(* Logix 5000 project; controller cal1632 1756-L62 rev 16.20; software revision 16.05; part 43 of 57 *)
(* tags used below, declared in another part *)
   FAULT : BOOL;
   HMI : BOOL;
   p01_recipe_active : recipe;
   p01r02_plc_scan_time_in_sec : REAL;
   p01r09_pb_global_reset : BOOL;
   p01r09_request_line_jog : BOOL;
   p01r09_stretch_mode : BOOL;
   p01r12_master_ramped_speed : REAL;
   p01r13_line_running : BOOL;
   p01r13_line_slow_ramp : BOOL;
   p01r13_permissive_drives : BOOL;
   p01r13_state : DINT;
   p02_real_from_hmi : hmi_real;
   p20r15_loa_on : BOOL;
   p20r16_lob_on : BOOL;
   p22r09_mode_thread : BOOL;
   p22r10_pid_psn : PID;
   p25_ai_speed : REAL;
   p25_ai_torque : REAL;
   p25_ai_ts2_lc : REAL;
   p25_ao_selected_speed : REAL;
   p25_ao_torque : REAL;
   p25_control_word : INT;
   p25_di_brake : BOOL;
   p25_di_jog : BOOL;
   p25_di_jog_fwd : BOOL;
   p25_di_jog_rev : BOOL;
   p25_di_run : BOOL;
   p25_di_therm : BOOL;
   p25_dint_to_hmi : DINT[16];
   p25_param_ts2_jog_speed : REAL;
   p25_status_word : INT;
   p25_ts2_acc_rate : REAL;
   p25_ts2_decel_rate : REAL;
   p25_ts2_vfd : ABB_PROTOCOL_VFD;
   p25r02_tension_dev_max : REAL;
   p25r02_tension_dev_min : REAL;
   p25r08 : routine;
   p25r08_timer_fault : TIMER[4];
   p25r08_timer_warning : TIMER[4];
   p25r09 : routine;
   p25r09_mode_jog : BOOL;
   p25r09_mode_run : BOOL;
   p25r09_mode_thread : BOOL;
   p25r09_pb_jog_fwd : BOOL;
   p25r09_pb_jog_rev : BOOL;
   p25r09_timer_fault : TIMER[4];
   p25r09_timer_warning : TIMER[4];
   p25r10 : routine;
   p25r10_calc_speed_offset : REAL;
   p25r10_param_psn_gain : REAL;
   p25r10_pid_manual_request : BOOL;
   p25r10_pid_out : REAL;
   p25r10_pid_psn : PID;
   p25r10_pid_psn_cv : REAL;
   p25r10_pid_psn_pv : REAL;
   p25r10_speed_offset : REAL;
   p25r10_tension_request : BOOL;
   p25r10_timer_fault : TIMER[4];
   p25r10_timer_warning : TIMER[4];
   p25r11 : routine;
   p25r11_acc_decel_ramp : SYS_ACC_DEC_RAMP;
   p25r11_at_zero : BOOL;
   p25r11_permissive_jog_thread : BOOL;
   p25r11_request_jog_fwd : BOOL;
   p25r11_request_jog_rev : BOOL;
   p25r11_request_line_jog : BOOL;
   p25r11_request_line_run : BOOL;
   p25r11_request_thread_fwd : BOOL;
   p25r11_request_thread_rev : BOOL;
   p25r11_selected_speed : REAL;
   p25r11_timer_fault : TIMER[10];
   p25r11_timer_warning : TIMER[4];
   p25r11_vfd_start_request : BOOL;
(* P25_Tension_Stand_2, continued *)

ROUTINE R08_Warnings   (* ladder *)
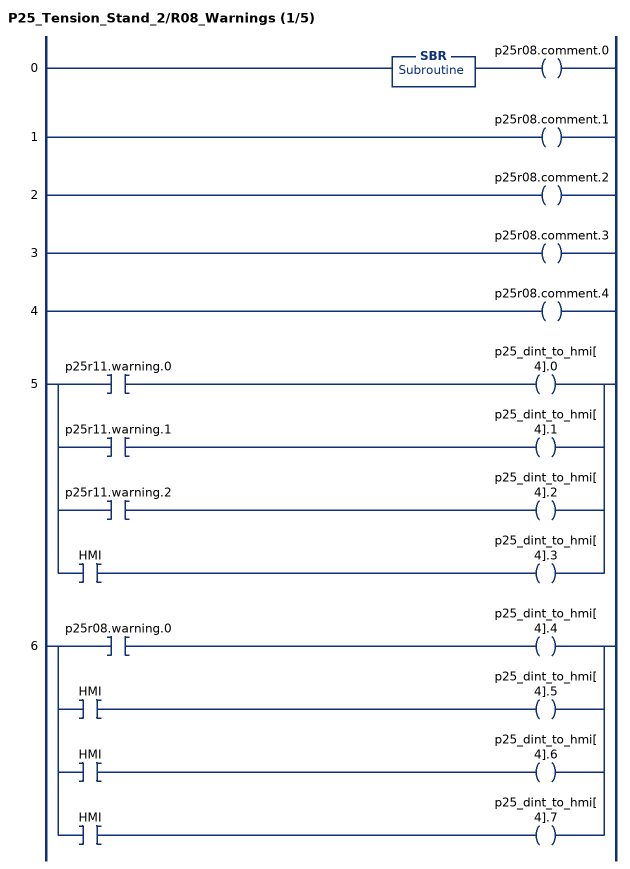
   0: SBR()OTE(p25r08.comment.0);
   1: OTE(p25r08.comment.1);
   2: OTE(p25r08.comment.2);
   3: OTE(p25r08.comment.3);
   4: OTE(p25r08.comment.4);
   5: [XIC(p25r11.warning.0) OTE(p25_dint_to_hmi[4].0) ,XIC(p25r11.warning.1) OTE(p25_dint_to_hmi[4].1) ,XIC(p25r11.warning.2) OTE(p25_dint_to_hmi[4].2) ,XIC(HMI) OTE(p25_dint_to_hmi[4].3) ];
   6: [XIC(p25r08.warning.0) OTE(p25_dint_to_hmi[4].4) ,XIC(HMI) OTE(p25_dint_to_hmi[4].5) ,XIC(HMI) OTE(p25_dint_to_hmi[4].6) ,XIC(HMI) OTE(p25_dint_to_hmi[4].7) ];
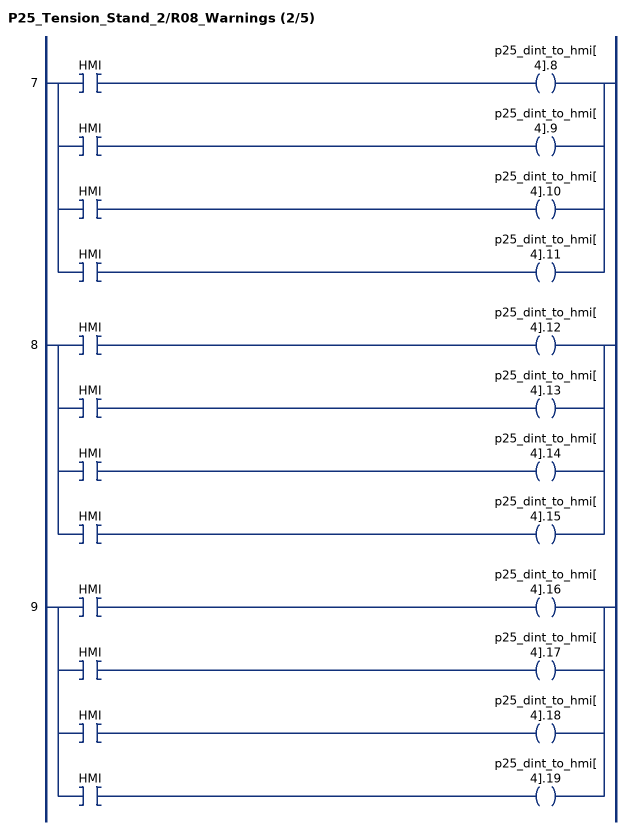
   7: [XIC(HMI) OTE(p25_dint_to_hmi[4].8) ,XIC(HMI) OTE(p25_dint_to_hmi[4].9) ,XIC(HMI) OTE(p25_dint_to_hmi[4].10) ,XIC(HMI) OTE(p25_dint_to_hmi[4].11) ];
   8: [XIC(HMI) OTE(p25_dint_to_hmi[4].12) ,XIC(HMI) OTE(p25_dint_to_hmi[4].13) ,XIC(HMI) OTE(p25_dint_to_hmi[4].14) ,XIC(HMI) OTE(p25_dint_to_hmi[4].15) ];
   9: [XIC(HMI) OTE(p25_dint_to_hmi[4].16) ,XIC(HMI) OTE(p25_dint_to_hmi[4].17) ,XIC(HMI) OTE(p25_dint_to_hmi[4].18) ,XIC(HMI) OTE(p25_dint_to_hmi[4].19) ];
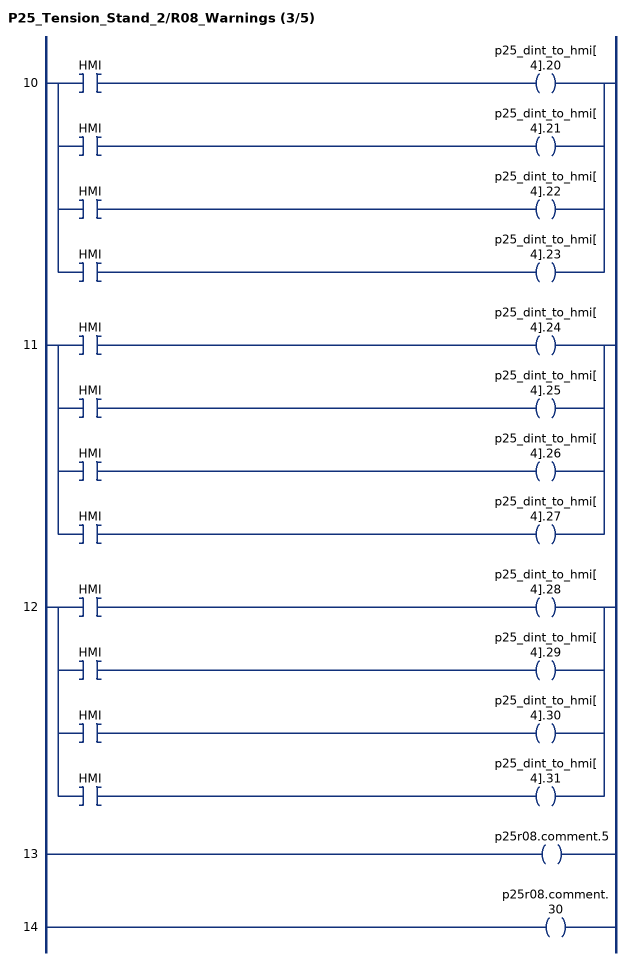
   10: [XIC(HMI) OTE(p25_dint_to_hmi[4].20) ,XIC(HMI) OTE(p25_dint_to_hmi[4].21) ,XIC(HMI) OTE(p25_dint_to_hmi[4].22) ,XIC(HMI) OTE(p25_dint_to_hmi[4].23) ];
   11: [XIC(HMI) OTE(p25_dint_to_hmi[4].24) ,XIC(HMI) OTE(p25_dint_to_hmi[4].25) ,XIC(HMI) OTE(p25_dint_to_hmi[4].26) ,XIC(HMI) OTE(p25_dint_to_hmi[4].27) ];
   12: [XIC(HMI) OTE(p25_dint_to_hmi[4].28) ,XIC(HMI) OTE(p25_dint_to_hmi[4].29) ,XIC(HMI) OTE(p25_dint_to_hmi[4].30) ,XIC(HMI) OTE(p25_dint_to_hmi[4].31) ];
   13: OTE(p25r08.comment.5);
   14: OTE(p25r08.comment.30);
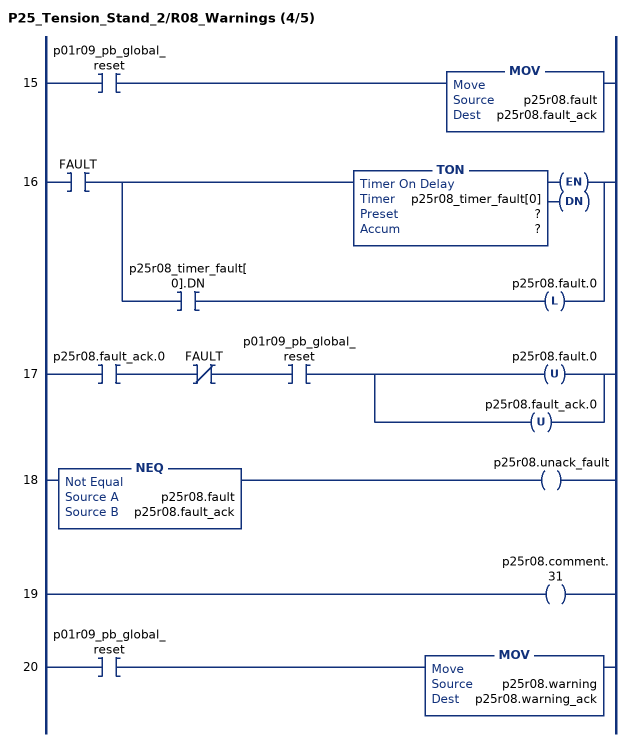
   15: XIC(p01r09_pb_global_reset)MOV(p25r08.fault,p25r08.fault_ack);
   16: XIC(FAULT)[TON(p25r08_timer_fault[0],?,?) ,XIC(p25r08_timer_fault[0].DN) OTL(p25r08.fault.0) ];
   17: XIC(p25r08.fault_ack.0)XIO(FAULT)XIC(p01r09_pb_global_reset)[OTU(p25r08.fault.0) ,OTU(p25r08.fault_ack.0) ];
   18: NEQ(p25r08.fault,p25r08.fault_ack)OTE(p25r08.unack_fault);
   19: OTE(p25r08.comment.31);
   20: XIC(p01r09_pb_global_reset)MOV(p25r08.warning,p25r08.warning_ack);
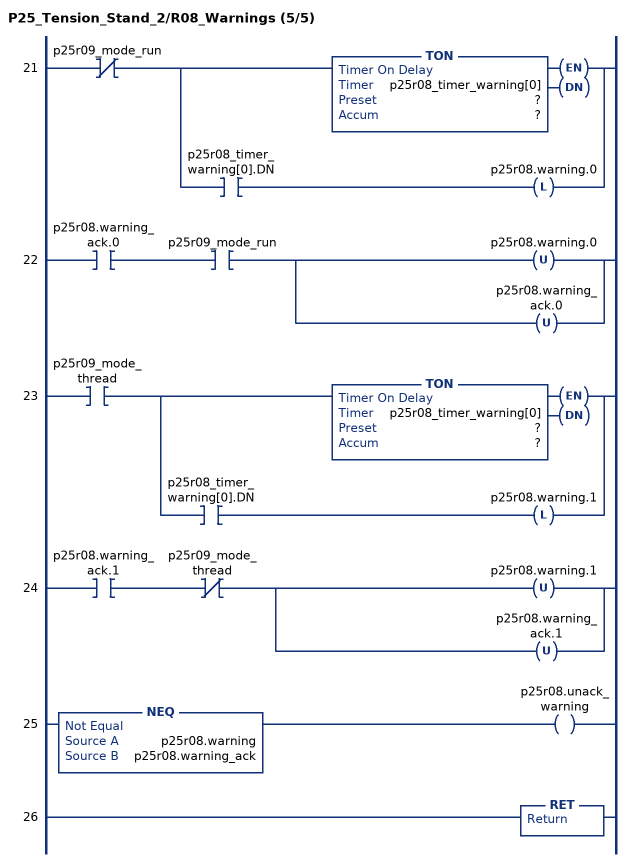
   21: XIO(p25r09_mode_run)[TON(p25r08_timer_warning[0],?,?) ,XIC(p25r08_timer_warning[0].DN) OTL(p25r08.warning.0) ];
   22: XIC(p25r08.warning_ack.0)XIC(p25r09_mode_run)[OTU(p25r08.warning.0) ,OTU(p25r08.warning_ack.0) ];
   23: XIC(p25r09_mode_thread)[TON(p25r08_timer_warning[0],?,?) ,XIC(p25r08_timer_warning[0].DN) OTL(p25r08.warning.1) ];
   24: XIC(p25r08.warning_ack.1)XIO(p25r09_mode_thread)[OTU(p25r08.warning.1) ,OTU(p25r08.warning_ack.1) ];
   25: NEQ(p25r08.warning,p25r08.warning_ack)OTE(p25r08.unack_warning);
   26: RET();
END_ROUTINE

ROUTINE R09_Modes   (* ladder *)
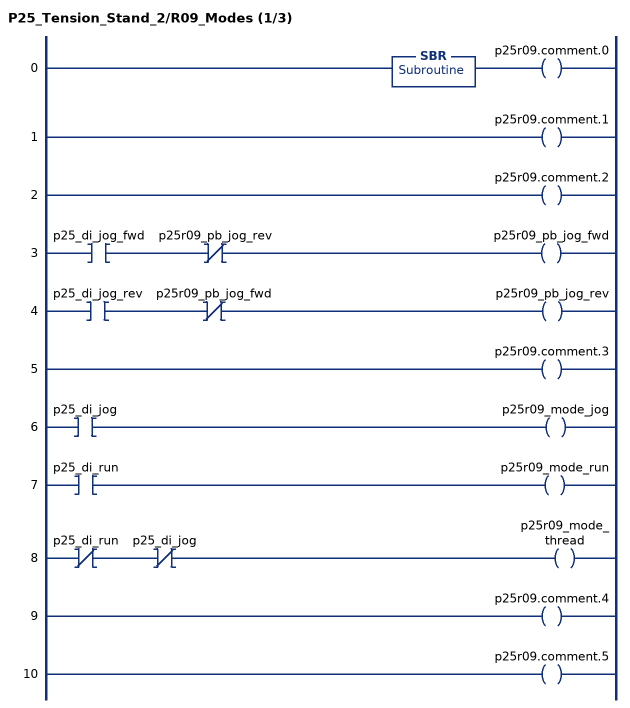
   0: SBR()OTE(p25r09.comment.0);
   1: OTE(p25r09.comment.1);
   2: OTE(p25r09.comment.2);
   3: XIC(p25_di_jog_fwd)XIO(p25r09_pb_jog_rev)OTE(p25r09_pb_jog_fwd);
   4: XIC(p25_di_jog_rev)XIO(p25r09_pb_jog_fwd)OTE(p25r09_pb_jog_rev);
   5: OTE(p25r09.comment.3);
   6: XIC(p25_di_jog)OTE(p25r09_mode_jog);
   7: XIC(p25_di_run)OTE(p25r09_mode_run);
   8: XIO(p25_di_run)XIO(p25_di_jog)OTE(p25r09_mode_thread);
   9: OTE(p25r09.comment.4);
   10: OTE(p25r09.comment.5);
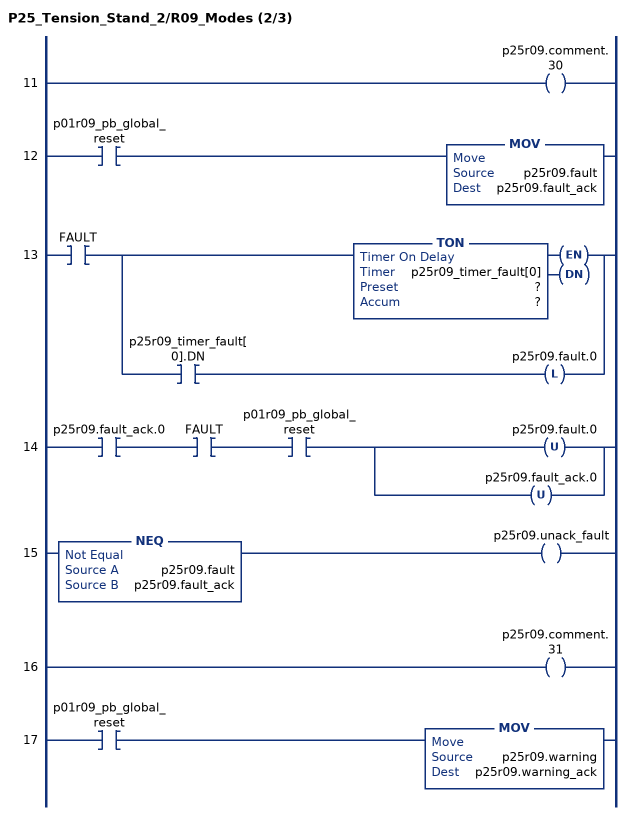
   11: OTE(p25r09.comment.30);
   12: XIC(p01r09_pb_global_reset)MOV(p25r09.fault,p25r09.fault_ack);
   13: XIC(FAULT)[TON(p25r09_timer_fault[0],?,?) ,XIC(p25r09_timer_fault[0].DN) OTL(p25r09.fault.0) ];
   14: XIC(p25r09.fault_ack.0)XIC(FAULT)XIC(p01r09_pb_global_reset)[OTU(p25r09.fault.0) ,OTU(p25r09.fault_ack.0) ];
   15: NEQ(p25r09.fault,p25r09.fault_ack)OTE(p25r09.unack_fault);
   16: OTE(p25r09.comment.31);
   17: XIC(p01r09_pb_global_reset)MOV(p25r09.warning,p25r09.warning_ack);
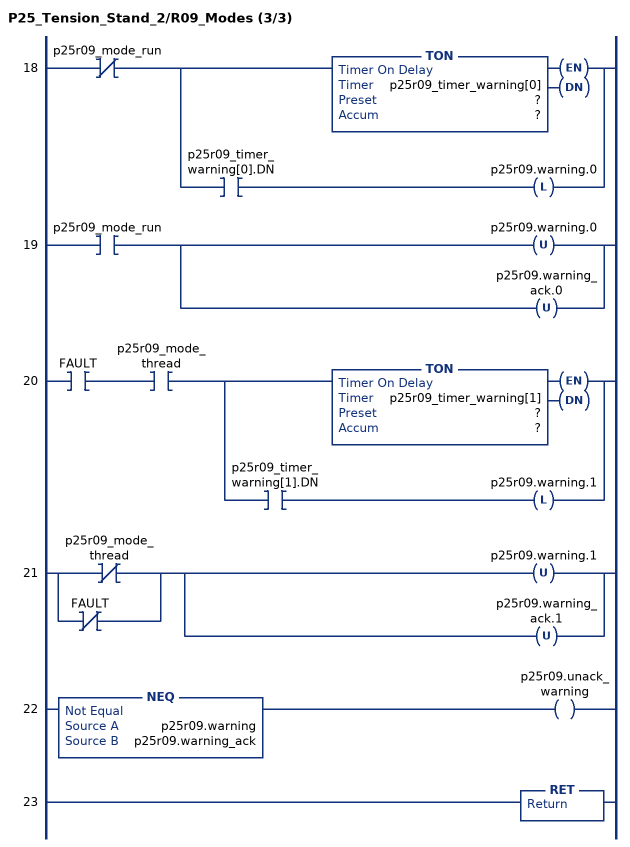
   18: XIO(p25r09_mode_run)[TON(p25r09_timer_warning[0],?,?) ,XIC(p25r09_timer_warning[0].DN) OTL(p25r09.warning.0) ];
   19: XIC(p25r09_mode_run)[OTU(p25r09.warning.0) ,OTU(p25r09.warning_ack.0) ];
   20: XIC(FAULT)XIC(p25r09_mode_thread)[TON(p25r09_timer_warning[1],?,?) ,XIC(p25r09_timer_warning[1].DN) OTL(p25r09.warning.1) ];
   21: [XIO(p25r09_mode_thread) ,XIO(FAULT) ][OTU(p25r09.warning.1) ,OTU(p25r09.warning_ack.1) ];
   22: NEQ(p25r09.warning,p25r09.warning_ack)OTE(p25r09.unack_warning);
   23: RET();
END_ROUTINE

ROUTINE R10_Speed_Control   (* ladder *)
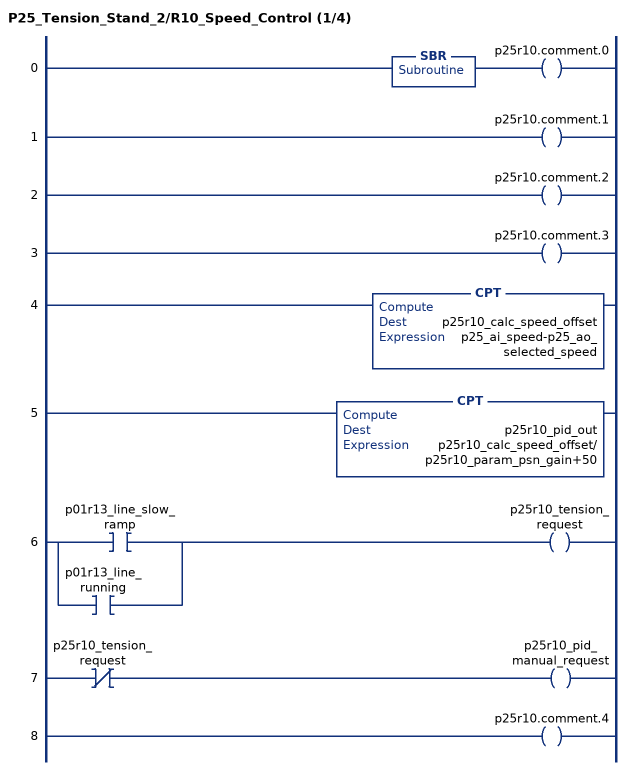
   0: SBR()OTE(p25r10.comment.0);
   1: OTE(p25r10.comment.1);
   2: OTE(p25r10.comment.2);
   3: OTE(p25r10.comment.3);
   4: CPT(p25r10_calc_speed_offset,p25_ai_speed-p25_ao_selected_speed);
   5: CPT(p25r10_pid_out,p25r10_calc_speed_offset/p25r10_param_psn_gain+50);
   6: [XIC(p01r13_line_slow_ramp) ,XIC(p01r13_line_running) ]OTE(p25r10_tension_request);
   7: XIO(p25r10_tension_request)OTE(p25r10_pid_manual_request);
   8: OTE(p25r10.comment.4);
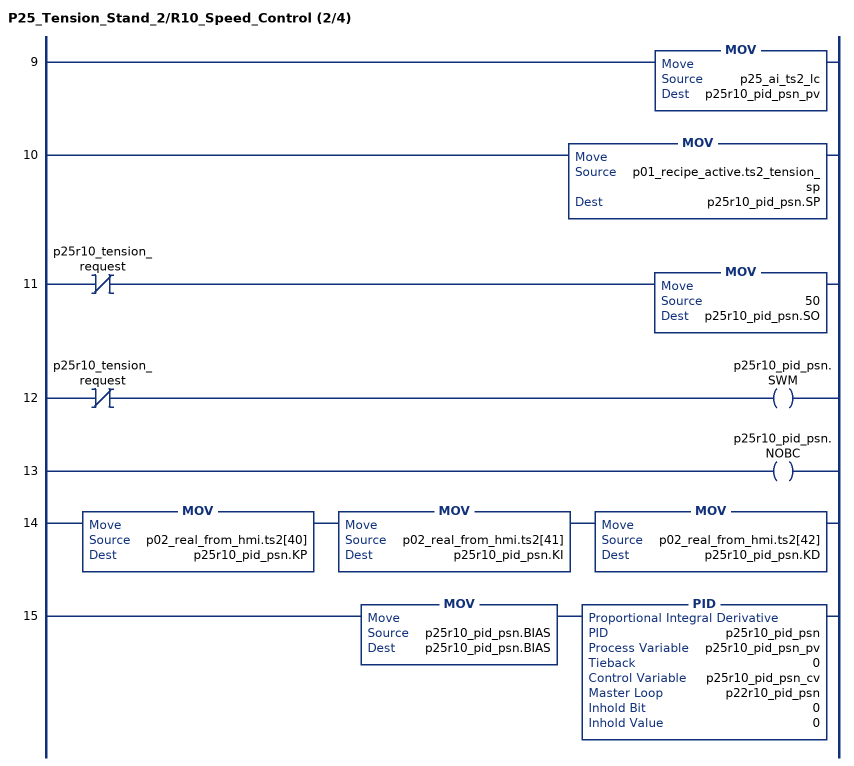
   9: MOV(p25_ai_ts2_lc,p25r10_pid_psn_pv);
   10: MOV(p01_recipe_active.ts2_tension_sp,p25r10_pid_psn.SP);
   11: XIO(p25r10_tension_request)MOV(50,p25r10_pid_psn.SO);
   12: XIO(p25r10_tension_request)OTE(p25r10_pid_psn.SWM);
   13: OTE(p25r10_pid_psn.NOBC);
   14: MOV(p02_real_from_hmi.ts2[40],p25r10_pid_psn.KP)MOV(p02_real_from_hmi.ts2[41],p25r10_pid_psn.KI)MOV(p02_real_from_hmi.ts2[42],p25r10_pid_psn.KD);
   15: MOV(p25r10_pid_psn.BIAS,p25r10_pid_psn.BIAS)PID(p25r10_pid_psn,p25r10_pid_psn_pv,0,p25r10_pid_psn_cv,p22r10_pid_psn,0,0);
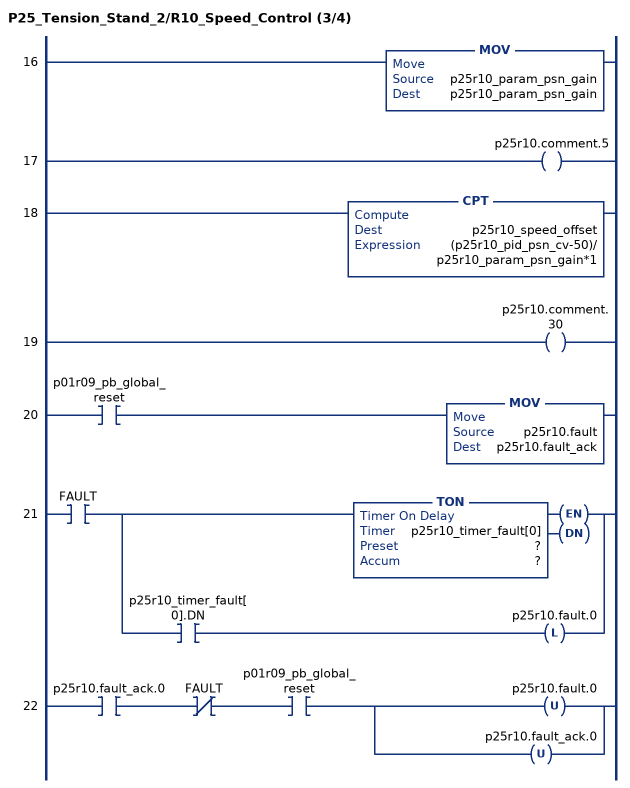
   16: MOV(p25r10_param_psn_gain,p25r10_param_psn_gain);
   17: OTE(p25r10.comment.5);
   18: CPT(p25r10_speed_offset,(p25r10_pid_psn_cv-50)/p25r10_param_psn_gain*1);
   19: OTE(p25r10.comment.30);
   20: XIC(p01r09_pb_global_reset)MOV(p25r10.fault,p25r10.fault_ack);
   21: XIC(FAULT)[TON(p25r10_timer_fault[0],?,?) ,XIC(p25r10_timer_fault[0].DN) OTL(p25r10.fault.0) ];
   22: XIC(p25r10.fault_ack.0)XIO(FAULT)XIC(p01r09_pb_global_reset)[OTU(p25r10.fault.0) ,OTU(p25r10.fault_ack.0) ];
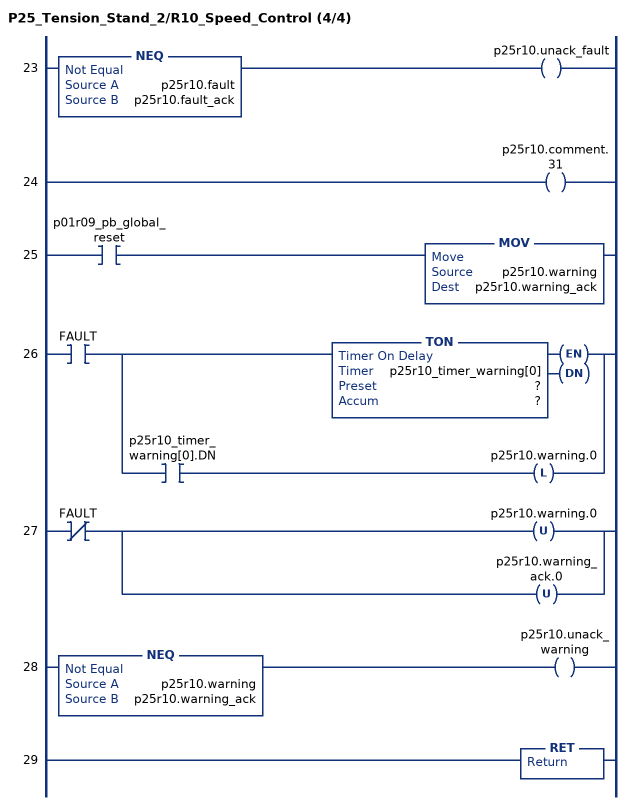
   23: NEQ(p25r10.fault,p25r10.fault_ack)OTE(p25r10.unack_fault);
   24: OTE(p25r10.comment.31);
   25: XIC(p01r09_pb_global_reset)MOV(p25r10.warning,p25r10.warning_ack);
   26: XIC(FAULT)[TON(p25r10_timer_warning[0],?,?) ,XIC(p25r10_timer_warning[0].DN) OTL(p25r10.warning.0) ];
   27: XIO(FAULT)[OTU(p25r10.warning.0) ,OTU(p25r10.warning_ack.0) ];
   28: NEQ(p25r10.warning,p25r10.warning_ack)OTE(p25r10.unack_warning);
   29: RET();
END_ROUTINE

ROUTINE R11_VFD   (* ladder *)
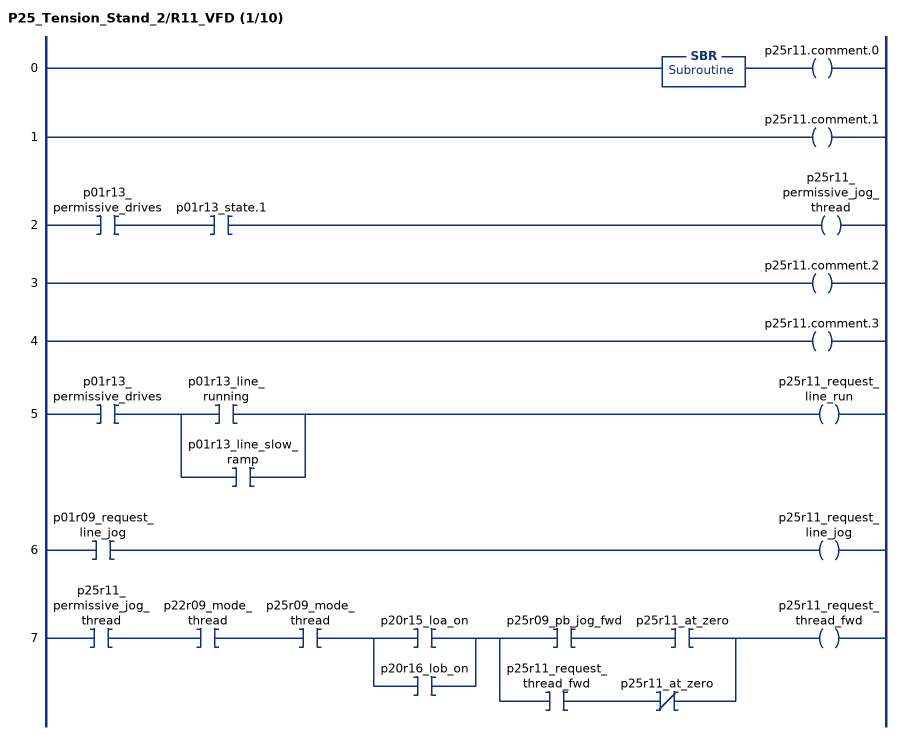
   0: SBR()OTE(p25r11.comment.0);
   1: OTE(p25r11.comment.1);
   2: XIC(p01r13_permissive_drives)XIC(p01r13_state.1)OTE(p25r11_permissive_jog_thread);
   3: OTE(p25r11.comment.2);
   4: OTE(p25r11.comment.3);
   5: XIC(p01r13_permissive_drives)[XIC(p01r13_line_running) ,XIC(p01r13_line_slow_ramp) ]OTE(p25r11_request_line_run);
   6: XIC(p01r09_request_line_jog)OTE(p25r11_request_line_jog);
   7: XIC(p25r11_permissive_jog_thread)XIC(p22r09_mode_thread)XIC(p25r09_mode_thread)[XIC(p20r15_loa_on) ,XIC(p20r16_lob_on) ][XIC(p25r09_pb_jog_fwd) XIC(p25r11_at_zero) ,XIC(p25r11_request_thread_fwd) XIO(p25r11_at_zero) ]OTE(p25r11_request_thread_fwd);
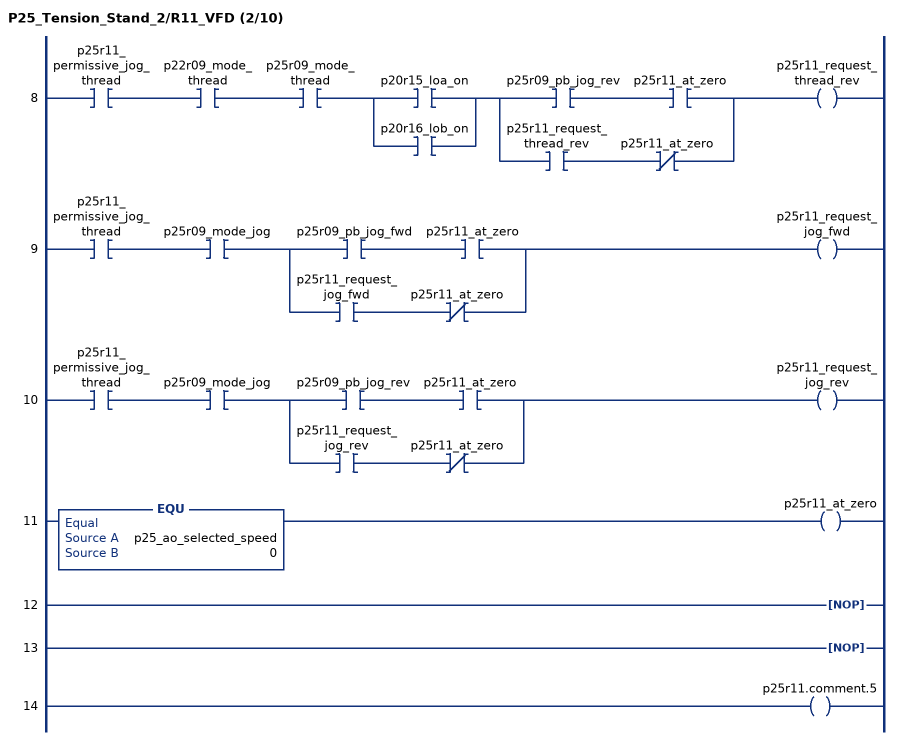
   8: XIC(p25r11_permissive_jog_thread)XIC(p22r09_mode_thread)XIC(p25r09_mode_thread)[XIC(p20r15_loa_on) ,XIC(p20r16_lob_on) ][XIC(p25r09_pb_jog_rev) XIC(p25r11_at_zero) ,XIC(p25r11_request_thread_rev) XIO(p25r11_at_zero) ]OTE(p25r11_request_thread_rev);
   9: XIC(p25r11_permissive_jog_thread)XIC(p25r09_mode_jog)[XIC(p25r09_pb_jog_fwd) XIC(p25r11_at_zero) ,XIC(p25r11_request_jog_fwd) XIO(p25r11_at_zero) ]OTE(p25r11_request_jog_fwd);
   10: XIC(p25r11_permissive_jog_thread)XIC(p25r09_mode_jog)[XIC(p25r09_pb_jog_rev) XIC(p25r11_at_zero) ,XIC(p25r11_request_jog_rev) XIO(p25r11_at_zero) ]OTE(p25r11_request_jog_rev);
   11: EQU(p25_ao_selected_speed,0)OTE(p25r11_at_zero);
   12: NOP();
   13: NOP();
   14: OTE(p25r11.comment.5);
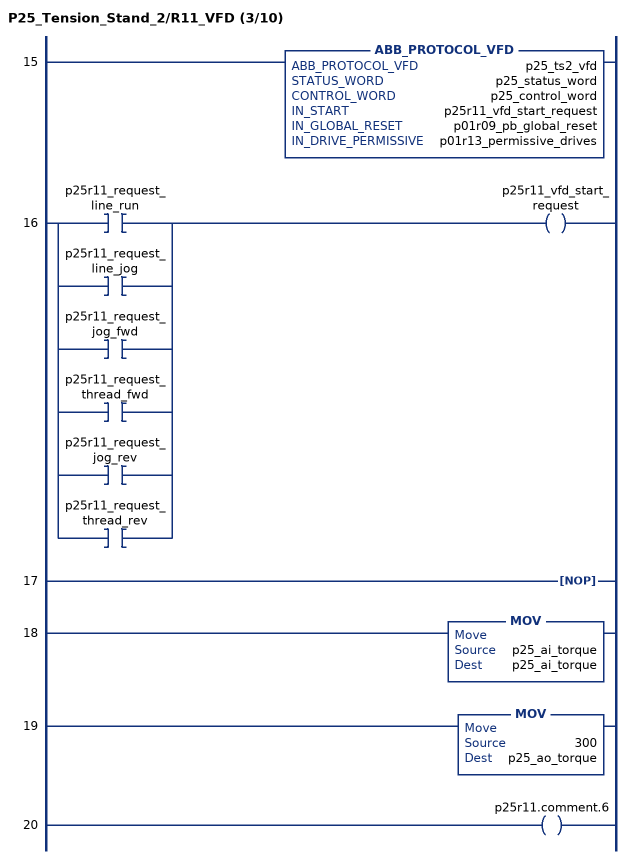
   15: ABB_PROTOCOL_VFD(p25_ts2_vfd,p25_status_word,p25_control_word,p25r11_vfd_start_request,p01r09_pb_global_reset,p01r13_permissive_drives);
   16: [XIC(p25r11_request_line_run) ,XIC(p25r11_request_line_jog) ,XIC(p25r11_request_jog_fwd) ,XIC(p25r11_request_thread_fwd) ,XIC(p25r11_request_jog_rev) ,XIC(p25r11_request_thread_rev) ]OTE(p25r11_vfd_start_request);
   17: NOP();
   18: MOV(p25_ai_torque,p25_ai_torque);
   19: MOV(300,p25_ao_torque);
   20: OTE(p25r11.comment.6);
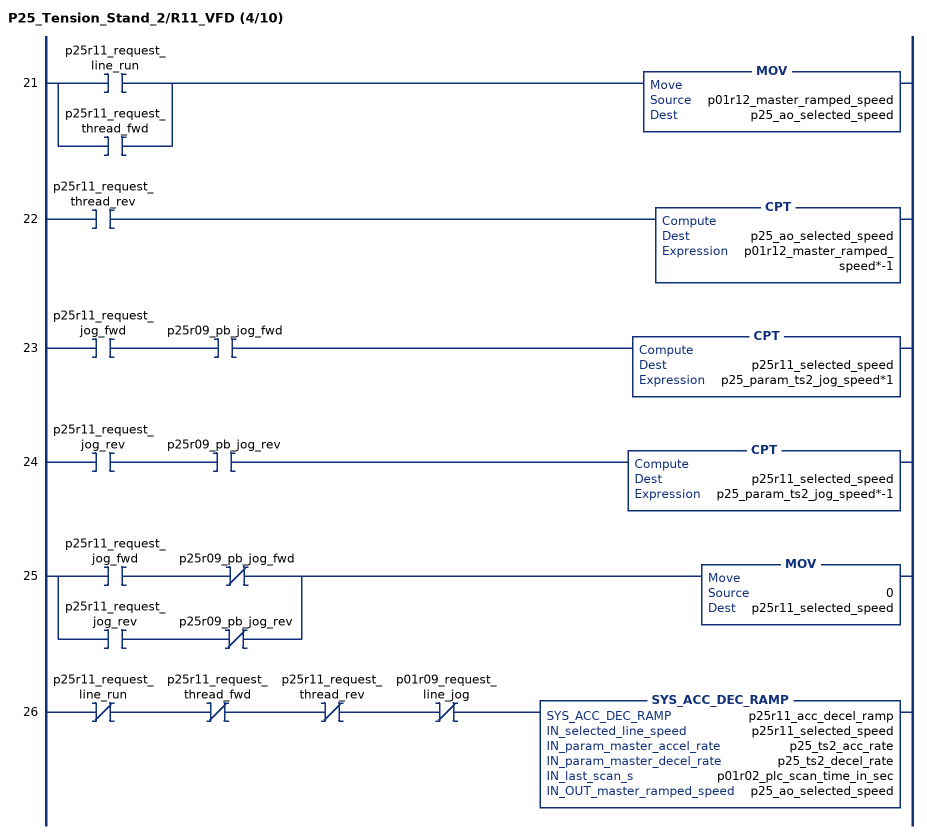
   21: [XIC(p25r11_request_line_run) ,XIC(p25r11_request_thread_fwd) ]MOV(p01r12_master_ramped_speed,p25_ao_selected_speed);
   22: XIC(p25r11_request_thread_rev)CPT(p25_ao_selected_speed,p01r12_master_ramped_speed*-1);
   23: XIC(p25r11_request_jog_fwd)XIC(p25r09_pb_jog_fwd)CPT(p25r11_selected_speed,p25_param_ts2_jog_speed*1);
   24: XIC(p25r11_request_jog_rev)XIC(p25r09_pb_jog_rev)CPT(p25r11_selected_speed,p25_param_ts2_jog_speed*-1);
   25: [XIC(p25r11_request_jog_fwd) XIO(p25r09_pb_jog_fwd) ,XIC(p25r11_request_jog_rev) XIO(p25r09_pb_jog_rev) ]MOV(0,p25r11_selected_speed);
   26: XIO(p25r11_request_line_run)XIO(p25r11_request_thread_fwd)XIO(p25r11_request_thread_rev)XIO(p01r09_request_line_jog)SYS_ACC_DEC_RAMP(p25r11_acc_decel_ramp,p25r11_selected_speed,p25_ts2_acc_rate,p25_ts2_decel_rate,p01r02_plc_scan_time_in_sec,p25_ao_selected_speed);
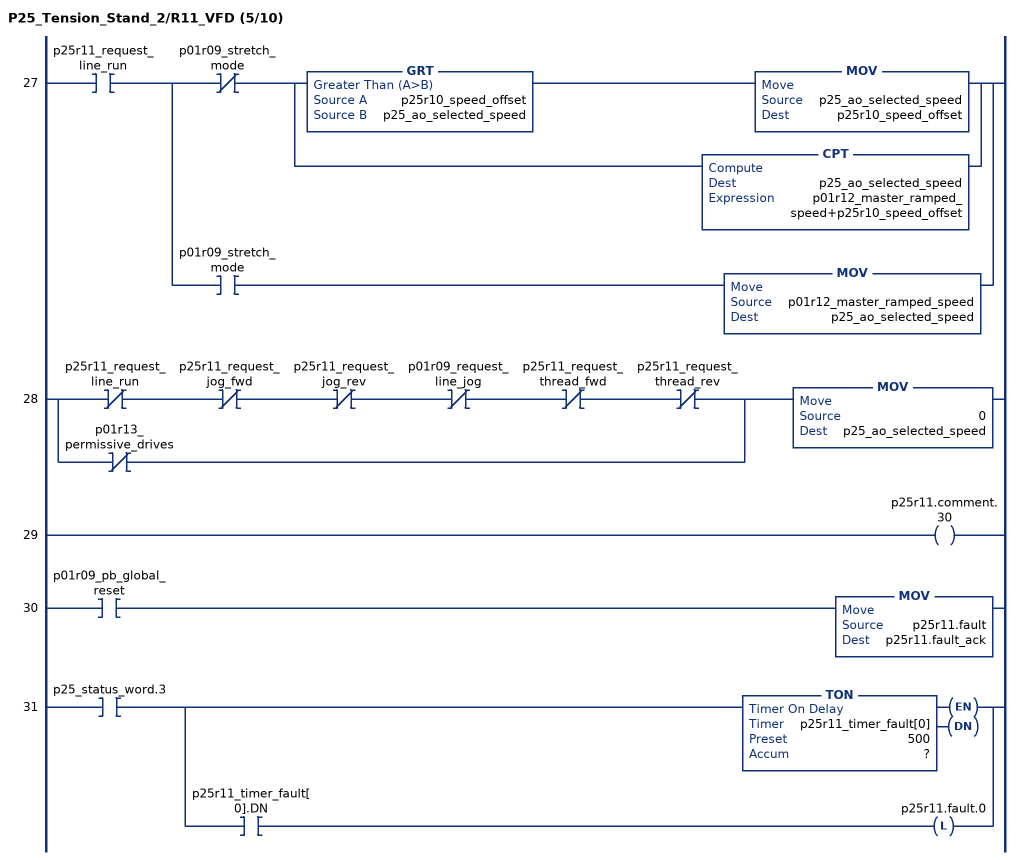
   27: XIC(p25r11_request_line_run)[XIO(p01r09_stretch_mode) [GRT(p25r10_speed_offset,p25_ao_selected_speed) MOV(p25_ao_selected_speed,p25r10_speed_offset) ,CPT(p25_ao_selected_speed,p01r12_master_ramped_speed+p25r10_speed_offset) ] ,XIC(p01r09_stretch_mode) MOV(p01r12_master_ramped_speed,p25_ao_selected_speed) ];
   28: [XIO(p25r11_request_line_run) XIO(p25r11_request_jog_fwd) XIO(p25r11_request_jog_rev) XIO(p01r09_request_line_jog) XIO(p25r11_request_thread_fwd) XIO(p25r11_request_thread_rev) ,XIO(p01r13_permissive_drives) ]MOV(0,p25_ao_selected_speed);
   29: OTE(p25r11.comment.30);
   30: XIC(p01r09_pb_global_reset)MOV(p25r11.fault,p25r11.fault_ack);
   31: XIC(p25_status_word.3)[TON(p25r11_timer_fault[0],?,?) ,XIC(p25r11_timer_fault[0].DN) OTL(p25r11.fault.0) ];
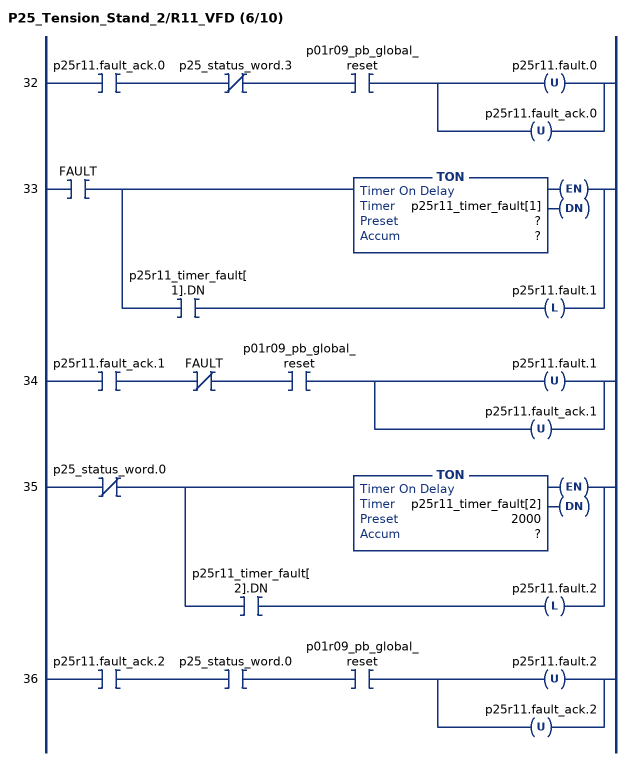
   32: XIC(p25r11.fault_ack.0)XIO(p25_status_word.3)XIC(p01r09_pb_global_reset)[OTU(p25r11.fault.0) ,OTU(p25r11.fault_ack.0) ];
   33: XIC(FAULT)[TON(p25r11_timer_fault[1],?,?) ,XIC(p25r11_timer_fault[1].DN) OTL(p25r11.fault.1) ];
   34: XIC(p25r11.fault_ack.1)XIO(FAULT)XIC(p01r09_pb_global_reset)[OTU(p25r11.fault.1) ,OTU(p25r11.fault_ack.1) ];
   35: XIO(p25_status_word.0)[TON(p25r11_timer_fault[2],?,?) ,XIC(p25r11_timer_fault[2].DN) OTL(p25r11.fault.2) ];
   36: XIC(p25r11.fault_ack.2)XIC(p25_status_word.0)XIC(p01r09_pb_global_reset)[OTU(p25r11.fault.2) ,OTU(p25r11.fault_ack.2) ];
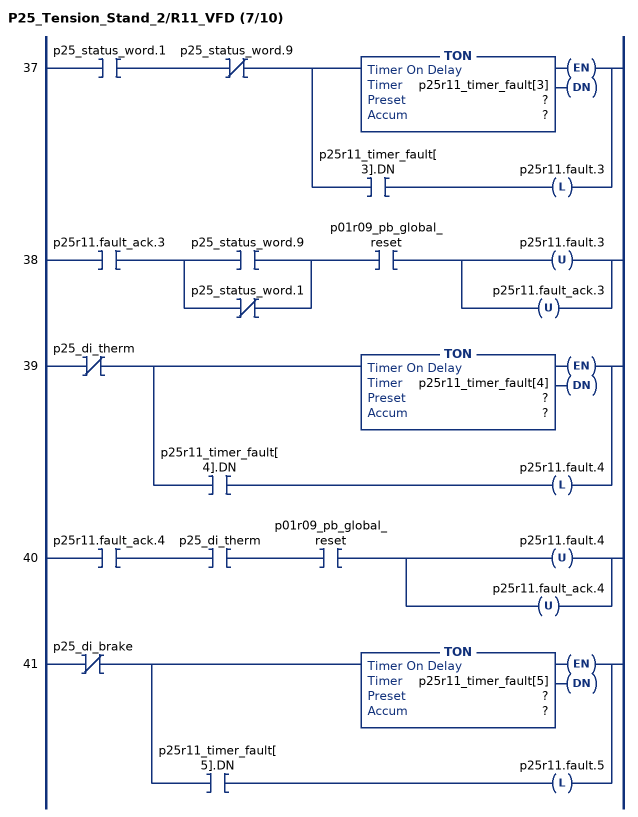
   37: XIC(p25_status_word.1)XIO(p25_status_word.9)[TON(p25r11_timer_fault[3],?,?) ,XIC(p25r11_timer_fault[3].DN) OTL(p25r11.fault.3) ];
   38: XIC(p25r11.fault_ack.3)[XIC(p25_status_word.9) ,XIO(p25_status_word.1) ]XIC(p01r09_pb_global_reset)[OTU(p25r11.fault.3) ,OTU(p25r11.fault_ack.3) ];
   39: XIO(p25_di_therm)[TON(p25r11_timer_fault[4],?,?) ,XIC(p25r11_timer_fault[4].DN) OTL(p25r11.fault.4) ];
   40: XIC(p25r11.fault_ack.4)XIC(p25_di_therm)XIC(p01r09_pb_global_reset)[OTU(p25r11.fault.4) ,OTU(p25r11.fault_ack.4) ];
   41: XIO(p25_di_brake)[TON(p25r11_timer_fault[5],?,?) ,XIC(p25r11_timer_fault[5].DN) OTL(p25r11.fault.5) ];
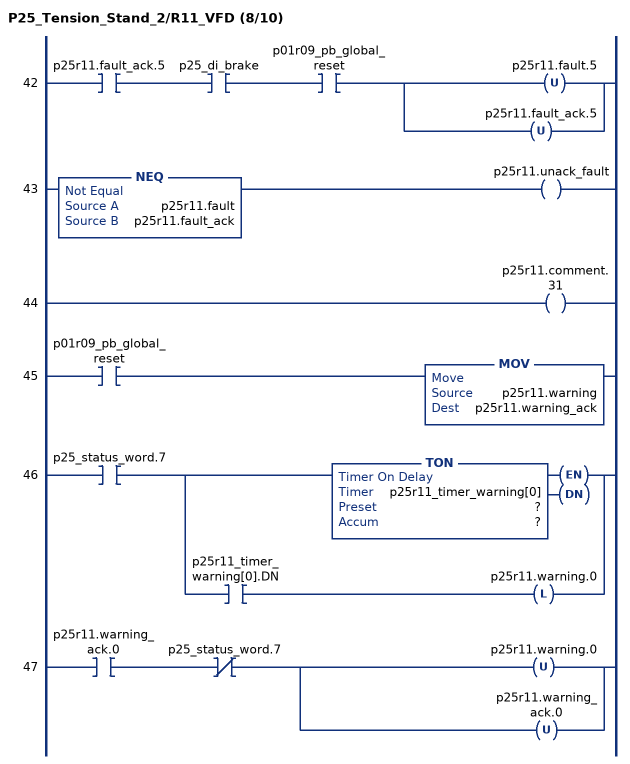
   42: XIC(p25r11.fault_ack.5)XIC(p25_di_brake)XIC(p01r09_pb_global_reset)[OTU(p25r11.fault.5) ,OTU(p25r11.fault_ack.5) ];
   43: NEQ(p25r11.fault,p25r11.fault_ack)OTE(p25r11.unack_fault);
   44: OTE(p25r11.comment.31);
   45: XIC(p01r09_pb_global_reset)MOV(p25r11.warning,p25r11.warning_ack);
   46: XIC(p25_status_word.7)[TON(p25r11_timer_warning[0],?,?) ,XIC(p25r11_timer_warning[0].DN) OTL(p25r11.warning.0) ];
   47: XIC(p25r11.warning_ack.0)XIO(p25_status_word.7)[OTU(p25r11.warning.0) ,OTU(p25r11.warning_ack.0) ];
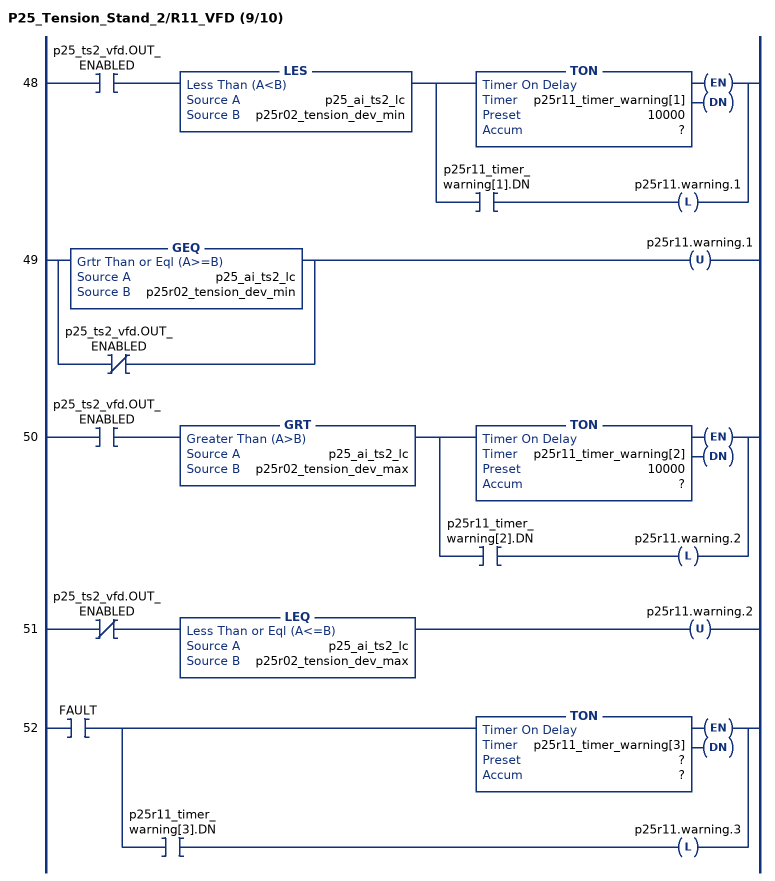
   48: XIC(p25_ts2_vfd.OUT_ENABLED)LES(p25_ai_ts2_lc,p25r02_tension_dev_min)[TON(p25r11_timer_warning[1],?,?) ,XIC(p25r11_timer_warning[1].DN) OTL(p25r11.warning.1) ];
   49: [GEQ(p25_ai_ts2_lc,p25r02_tension_dev_min) ,XIO(p25_ts2_vfd.OUT_ENABLED) ]OTU(p25r11.warning.1);
   50: XIC(p25_ts2_vfd.OUT_ENABLED)GRT(p25_ai_ts2_lc,p25r02_tension_dev_max)[TON(p25r11_timer_warning[2],?,?) ,XIC(p25r11_timer_warning[2].DN) OTL(p25r11.warning.2) ];
   51: XIO(p25_ts2_vfd.OUT_ENABLED)LEQ(p25_ai_ts2_lc,p25r02_tension_dev_max)OTU(p25r11.warning.2);
   52: XIC(FAULT)[TON(p25r11_timer_warning[3],?,?) ,XIC(p25r11_timer_warning[3].DN) OTL(p25r11.warning.3) ];
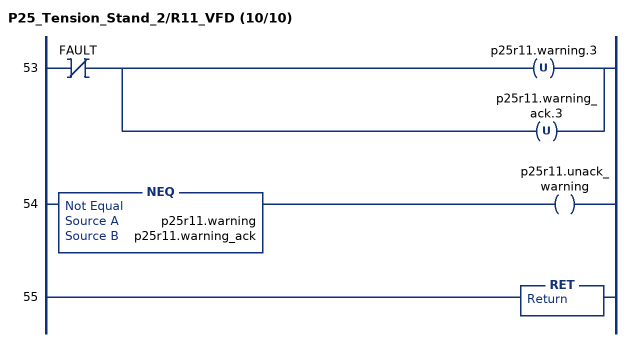
   53: XIO(FAULT)[OTU(p25r11.warning.3) ,OTU(p25r11.warning_ack.3) ];
   54: NEQ(p25r11.warning,p25r11.warning_ack)OTE(p25r11.unack_warning);
   55: RET();
END_ROUTINE
END_PROGRAM
